TYPE ST_RV_les_Zustand :
STRUCT
	Stellung				: USINT;
END_STRUCT
END_TYPE

(* stored: Version 1.1.0.1, ProductVersion 3.1.4024.9
   DUT ST_RV_les_Zustand: Id {c65105cb-61f8-462e-a5e5-06d29de14e7b} *)
